(* CoDeSys 2.3 export: ST_VALVE_BAR.EXP *)

(* Data type *)
TYPE ST_VALVE_BAR :
STRUCT
	Name : STRING;

	Bar : REAL;
	mA  : UINT;

	(*Calib*)
	Cal_K   : REAL;
	Cal_Off : REAL;

END_STRUCT
END_TYPE
